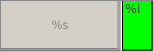
VISUALIZATION VISU_FCTS_SA  // 154x52
VAR_INPUT
	m_Input_ID_XML: UDINT;
END_VAR
VAR_IN_OUT
	m_Input_Operation:	BLOCK_OPERATION;
END_VAR
VAR_INPUT
	m_Input_UserRight:	BOOL;
END_VAR
    Button (0,0 120x50), "%s", invisible if: NOT m_Input_Operation.AUTOR_IHM OR NOT m_Input_UserRight, text list: 'TextList_SA_Operations', text index: m_Input_ID_XML
        toggle m_Input_Operation.ON_IHM
    RoundedRectangle (122,0 30x50), "%i", text variable: m_Input_Operation.STATUS, invisible if: NOT m_Input_Operation.AR
    Button (0,0 120x50), "%s", invisible if: m_Input_Operation.AUTOR_IHM AND m_Input_UserRight, text list: 'TextList_SA_Operations', text index: m_Input_ID_XML
    RoundedRectangle (122,0 30x50), "%i", text variable: m_Input_Operation.STATUS, invisible if: NOT m_Input_Operation.EC
    RoundedRectangle (122,0 30x50), "%i", text variable: m_Input_Operation.STATUS, invisible if: NOT m_Input_Operation.OK
END_VISUALIZATION

(* stored: Version 1.1.0.1, ProductVersion 3.1.4024.10
   Visu VISU_FCTS_SA: Id {a22fd1a4-67ad-4b40-8e08-b822dd17867e} *)
